FUNCTION_BLOCK Conveyor
VAR
	position : REAL;
	velocity : REAL;
	
	retracted : BOOL; //vertical conveyors
END_VAR

METHOD backward : BOOL
VAR_INPUT
END_VAR
END_METHOD

METHOD extend : BOOL
VAR_INPUT
END_VAR
END_METHOD

METHOD forward : BOOL
VAR_INPUT
END_VAR
END_METHOD

METHOD getPosition : REAL;
VAR_INPUT
END_VAR
getPosition := position;
END_METHOD

METHOD getVelocity : REAL;
VAR_INPUT
END_VAR
getVelocity := velocity;
END_METHOD

METHOD reset : BOOL
VAR_INPUT
END_VAR
position := 0;
velocity := velocity; //no change

extend();
END_METHOD

METHOD retract : BOOL
VAR_INPUT
END_VAR
END_METHOD

METHOD target : BOOL
VAR_INPUT
	targetPosition : REAL;
END_VAR
END_METHOD

END_FUNCTION_BLOCK

(* stored: Version 1.1.0.1, ProductVersion 3.1.4024.11
   POU Conveyor: Id {de162f93-5907-4a07-a0b5-f0d4a4560d6a}, SpecialFunc None
   Method backward: Id {86f9a8ba-67b5-4107-b253-01b957c1bf10}
   Method extend: Id {8f868bfa-a538-4183-8601-28b224890cc0}
   Method forward: Id {87d44885-25ee-41d2-af0e-9e2311376d2b}
   Method getPosition: Id {0a57e989-d05e-48a8-a083-297204d36b31}
   Method getVelocity: Id {0f80eae4-24a1-473c-ab6f-d7f6b6e5b700}
   Method reset: Id {d40da114-e5c3-466f-8119-1749f88356bf}
   Method retract: Id {e67cd767-48c0-4514-8169-49f3436776ec}
   Method target: Id {ea17b475-eaf3-4273-b8f8-a97119ee998d} *)
